{attribute 'qualified_only'}
VAR_GLOBAL
	POWER_ON : BOOL;
    Auto_mode: BOOL;
	Manual_Mode: BOOL;
	TEMP : BOOL;
	
	
	M_CC1_CLAMPING_UNIT1_3_WP : BOOL;
	M_CC1_CLAMPING_UNIT1_3_HP : BOOL;
	M_CC2_CLAMPING_UNIT2_3_WP : BOOL;
	M_CC2_CLAMPING_UNIT2_3_HP : BOOL;
	M_CC3_CLAMPING_UNIT3_3_WP : BOOL;
	M_CC3_CLAMPING_UNIT3_3_HP : BOOL;
	M_CC4_CLAMPING_UNIT4_3_WP : BOOL;
	M_CC4_CLAMPING_UNIT4_3_HP : BOOL;
	M_CC5_CLAMPING_UNIT5_1_WP : BOOL;
	M_CC5_CLAMPING_UNIT5_1_HP : BOOL;
	M_CC6_CLAMPING_UNIT6_1_WP : BOOL;
	M_CC6_CLAMPING_UNIT6_1_HP : BOOL;
    A_CC1_CLAMPING_UNIT1_3_WP : BOOL;
	A_CC1_CLAMPING_UNIT1_3_HP : BOOL;
	A_CC2_CLAMPING_UNIT2_3_WP : BOOL;
	A_CC2_CLAMPING_UNIT2_3_HP : BOOL;
	A_CC3_CLAMPING_UNIT3_3_WP : BOOL;
	A_CC3_CLAMPING_UNIT3_3_HP : BOOL;
	A_CC4_CLAMPING_UNIT4_3_WP : BOOL;
	A_CC4_CLAMPING_UNIT4_3_HP : BOOL;
	A_CC5_CLAMPING_UNIT5_1_WP : BOOL;
	A_CC5_CLAMPING_UNIT5_1_HP : BOOL;
	A_CC6_CLAMPING_UNIT6_1_WP : BOOL;
	A_CC6_CLAMPING_UNIT6_1_HP : BOOL;
	TEMP_CC1_WP_FEEDBACK : BOOL;
	TEMP_CC1_HP_FEEDBACK : BOOL;
	TEMP_CC2_WP_FEEDBACK : BOOL;
	TEMP_CC2_HP_FEEDBACK : BOOL;
	TEMP_CC3_WP_FEEDBACK : BOOL;
	TEMP_CC3_HP_FEEDBACK : BOOL;
	TEMP_CC4_WP_FEEDBACK : BOOL;
	TEMP_CC4_HP_FEEDBACK : BOOL;
	TEMP_CC5_WP_FEEDBACK : BOOL;
	TEMP_CC5_HP_FEEDBACK : BOOL;
	TEMP_CC6_WP_FEEDBACK : BOOL;
	TEMP_CC6_HP_FEEDBACK : BOOL;
	A_FIX1_ALL_CLAMP_WORK : BOOL;
	A_FIX1_ALL_CLAMP_HOME : BOOL;
	A_FIX2_ALL_CLAMP_WORK : BOOL;
	A_FIX2_ALL_CLAMP_HOME : BOOL;
	M_FIX1_ALL_CLAMP_HOME_PB : BOOL;
	//SENSOR
	A_FIX1_PART_1ST : BOOL;
	A_FIX1_PART_2ND : BOOL;
	A_FIX1_PART_3RD : BOOL;
	A_FIX1_PART_4TH : BOOL;
	A_FIX1_PART_5TH : BOOL;
	A_FIX1_PART_6TH : BOOL;
	A_FIX2_PART_1ST : BOOL;
	A_FIX2_PART_2ND : BOOL;
	A_FIX2_PART_3RD : BOOL;
	A_FIX2_PART_4TH : BOOL;
	A_FIX2_PART_5TH : BOOL;
	A_FIX2_PART_6TH : BOOL;
	// TT POSITION
	M_1ST_POSITION_TT_CMD : BOOL;
	M_2ND_POSITION_TT_CMD : BOOL;
	A_1ST_POSITION_TT_CMD : BOOL;
	A_2ND_POSITION_TT_CMD : BOOL;
	A_FEEDBACK_TT_FWD : BOOL;
	A_FEEDBACK_TT_REV : BOOL;
	// Trunion POSITION
	A_Clamp_ok : BOOL;
	M_Fwd_POSITION : BOOL;
	M_Rev_POSITION : BOOL;
	A_Fwd_POSITION : BOOL;
	A_Rev_POSITION : BOOL;
	A_FEEDBACK_TRUNION_FWD : BOOL;
	A_FEEDBACK_TRUNION_REV : BOOL;
	//ROLLER DOOR
	M_Roll_Dr_Open  : BOOL;
	M_Roll_Dr_Close : BOOL;
	A_Open_CMD      : BOOL;
    A_Close_CMD     : BOOL;
	A_Safety_Beam : BOOL;
	A_FEEDBACK_RD_OPEN : BOOL;
	A_FEEDBACK_RD_CLOSE : BOOL;
	//ROBOT
	ROBOT_START : BOOL;
	SAFETY_OK : BOOL;
	ROBOT_JOG : BOOL;
	ROBOT_COMPLETE : BOOL;
	ROBOT_BUSY : BOOL;
	ROBOT_HOME : BOOL;
	TEMP_ROB : BOOL;
	//MH_ROBOT
	MH_ROBOT_START : BOOL;
	MH_SAFETY_OK : BOOL;
	MH_ROBOT_JOG : BOOL;
	MH_ROBOT_COMPLETE : BOOL;
	MH_ROBOT_BUSY : BOOL;
	MH_ROBOT_HOME : BOOL;
	MH_TEMP_ROB : BOOL;
	
	
	
END_VAR

(* stored: Version 1.1.0.1, ProductVersion 3.1.4024.16
   GVL OP_Memory_DB: Id {bf9a8e60-94bf-48be-9318-80bc80477e33} *)
